// TIA Portal project "PumpProject" (V16)

(* hardware
DEVICE "S7-1200 station_1"  S7-1200 Station
   slot 0: "Rack_0"  S7-1200 Rack  Rack  V1.0
   slot 1: "PLC_1"  CPU 1214C DC/DC/DC  6ES7 214-1AG40-0XB0  V4.0
   slot 3: "AQ 1x12BIT_1"  AQ1 signal board  6ES7 232-4HA30-0XB0  V1.0
*)

// ===== PLC "PLC_1"  CPU 1214C DC/DC/DC =====

VAR_GLOBAL   // PLC tag table "Default tag table"
   "MoreButton" AT %M0.0 : Bool;
   "More" AT %M0.1 : Bool;
   "Less" AT %M0.2 : Bool;
   "LessButton" AT %M0.3 : Bool;
   "StartP1" AT %M0.4 : Bool;
   "StopP1" AT %M0.5 : Bool;
   "StartP2" AT %M0.6 : Bool;
   "StopP2" AT %M0.7 : Bool;
   "StartP3" AT %M1.0 : Bool;
   "StopP3" AT %M1.1 : Bool;
   "comP1" AT %MB2 : Byte;
   "testslay" AT %Q0.0 : Bool;
   "testsalw" AT %M1.2 : Bool;
   "RestOff" AT %M1.3 : Bool;
   "RestOn" AT %M1.4 : Bool;
   "Counter1Off" AT %M1.5 : Bool;
   "Counter2Off" AT %M1.6 : Bool;
   "MStart" AT %M1.7 : Bool;
   "MStop" AT %M3.0 : Bool;
END_VAR

// folder: System blocks/Program resources

DATA_BLOCK "OnPumpM"   // DB1
{ S7_Optimized_Access := 'TRUE' }
AUTHOR : Simatic
FAMILY : IEC
NAME : CNTR
VERSION : 1.0
// stored: InstanceOfName IEC_COUNTER
"IEC_COUNTER"
BEGIN
END_DATA_BLOCK

DATA_BLOCK "OnPump"   // DB2
{ S7_Optimized_Access := 'TRUE' }
AUTHOR : Simatic
FAMILY : IEC
NAME : CNTR
VERSION : 1.0
// stored: InstanceOfName IEC_COUNTER
"IEC_COUNTER"
BEGIN
END_DATA_BLOCK

DATA_BLOCK "OffPump"   // DB3
{ S7_Optimized_Access := 'TRUE' }
AUTHOR : Simatic
FAMILY : IEC
NAME : CNTR
VERSION : 1.0
// stored: InstanceOfName IEC_COUNTER
"IEC_COUNTER"
BEGIN
END_DATA_BLOCK

DATA_BLOCK "OffPumpM"   // DB4
{ S7_Optimized_Access := 'TRUE' }
AUTHOR : Simatic
FAMILY : IEC
NAME : CNTR
VERSION : 1.0
// stored: InstanceOfName IEC_COUNTER
"IEC_COUNTER"
BEGIN
END_DATA_BLOCK

// folder: (top level)

ORGANIZATION_BLOCK "Main"   // OB1, LAD, ProgramCycle
TITLE = "Main Program Sweep (Cycle)"
{ S7_Optimized_Access := 'TRUE' }
VERSION : 0.1
   VAR_INPUT
      Initial_Call : Bool;   // Initial call of this OB
      Remanence : Bool;   // =True, if remanent data are available
   END_VAR
   VAR_TEMP
      ResetOn : Bool;
   END_VAR
BEGIN

REGION Network 1
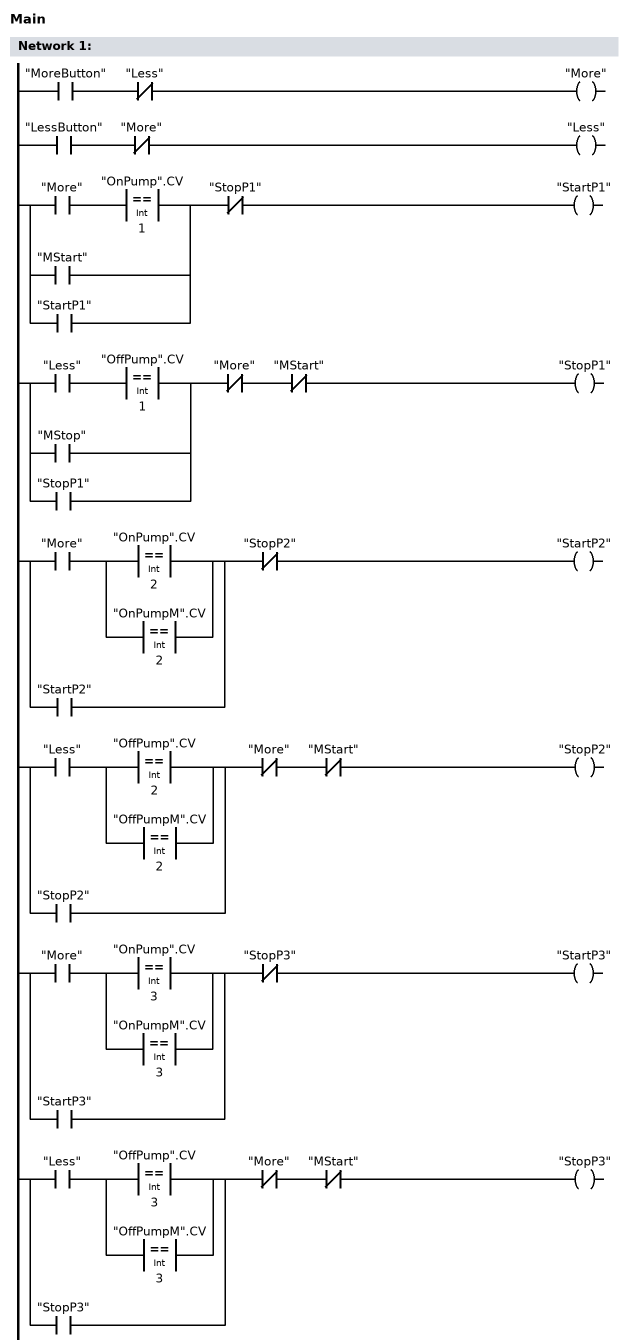
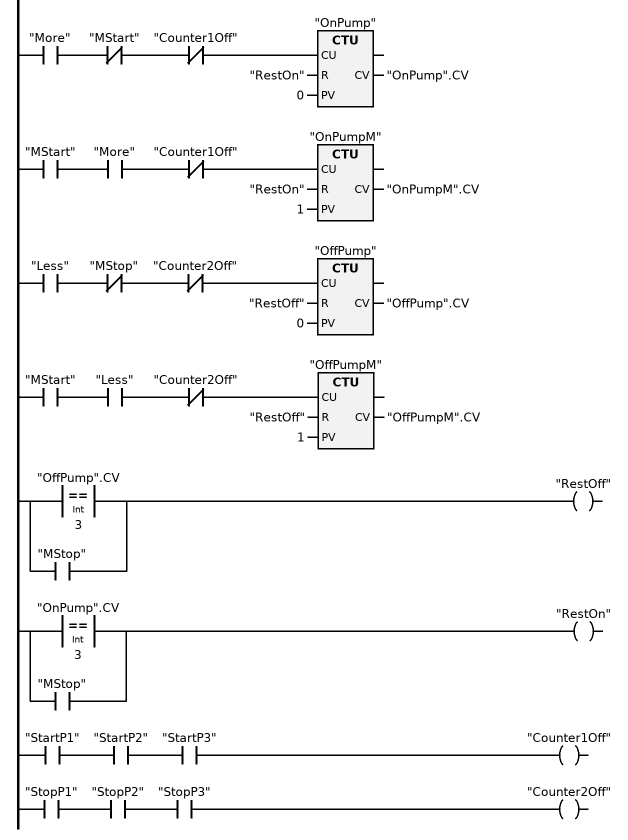
   "More" := "MoreButton" AND NOT "Less";
   "Less" := "LessButton" AND NOT "More";
   "StartP1" := (("More" AND ("OnPump".CV = 1)) OR "MStart" OR "StartP1") AND NOT "StopP1";
   "StopP1" := (("Less" AND ("OffPump".CV = 1)) OR "MStop" OR "StopP1") AND NOT "More" AND NOT "MStart";
   "StartP2" := (("More" AND (("OnPump".CV = 2) OR ("OnPumpM".CV = 2))) OR "StartP2") AND NOT "StopP2";
   "StopP2" := (("Less" AND (("OffPump".CV = 2) OR ("OffPumpM".CV = 2))) OR "StopP2") AND NOT "More" AND NOT "MStart";
   "StartP3" := (("More" AND (("OnPump".CV = 3) OR ("OnPumpM".CV = 3))) OR "StartP3") AND NOT "StopP3";
   "StopP3" := (("Less" AND (("OffPump".CV = 3) OR ("OffPumpM".CV = 3))) OR "StopP3") AND NOT "More" AND NOT "MStart";
   "OnPump".CTU(CU := "More" AND NOT "MStart" AND NOT "Counter1Off", R := "RestOn", PV := 0, CV => "OnPump".CV);
   "OnPumpM".CTU(CU := "MStart" AND "More" AND NOT "Counter1Off", R := "RestOn", PV := 1, CV => "OnPumpM".CV);
   "OffPump".CTU(CU := "Less" AND NOT "MStop" AND NOT "Counter2Off",
                 R := "RestOff",
                 PV := 0,
                 CV => "OffPump".CV);
   "OffPumpM".CTU(CU := "MStart" AND "Less" AND NOT "Counter2Off", R := "RestOff", PV := 1, CV => "OffPumpM".CV);
   "RestOff" := ("OffPump".CV = 3) OR "MStop";
   "RestOn" := ("OnPump".CV = 3) OR "MStop";
   "Counter1Off" := "StartP1" AND "StartP2" AND "StartP3";
   "Counter2Off" := "StopP1" AND "StopP2" AND "StopP3";
END_REGION
END_ORGANIZATION_BLOCK